{attribute 'qualified_only'}
{attribute 'strict'}
{attribute 'to_string'}
TYPE E_SystemState  :
(
    eState_Init := 0,
    eState_Manual,
    eState_AutoIdle,
	eState_AutoRunning,
	eState_Error
);
END_TYPE

(* stored: Version 1.1.0.1
   DUT E_SystemState: Id {b75c3681-1d71-4644-a7d7-6a544b63d96a} *)
